Fanuc KAREL source: kf00004.KL

-- PROVISIONAL review KL for V940-1; original PC SHA256 2f02e9247c93bcc4ce6be4374bce4bc9104b2ce51b48f90a11b16b7b15de6204
-- Incomplete behavior may be omitted. Consult companion uncertainty JSON. Do not deploy.
PROGRAM KF00004
%NOLOCKGROUP
VAR
  I : INTEGER
  J : INTEGER
  X : REAL
  Y : REAL
  B : BOOLEAN
  C : BOOLEAN
  TXT : STRING[80]
  TXT2 : STRING[80]
  STATUS : INTEGER
-- UNRESOLVED_DECL AI type=002010
-- UNRESOLVED_DECL BI type=002010
-- UNRESOLVED_DECL P type=000102
-- UNRESOLVED_DECL JP type=000199
-- UNRESOLVED_DECL PF type=000101
-- UNRESOLVED_DECL V1 type=000013
-- UNRESOLVED_DECL V2 type=000013
BEGIN
  -- V9_ZERO_TABLE_METADATA_HINT layout=0001; no indexed target words; source/name/runtime held
  -- UNRESOLVED_PC offsets 5-16; opcodes 2E,23
  -- UNRESOLVED_PC offsets 21-32; opcodes 2E,23
  -- UNRESOLVED_PC offsets 37-56; opcodes 21,21,55,23
  -- UNRESOLVED_PC offsets 61-65; opcodes 7F
END KF00004
